FUNCTION_BLOCK FB_DiagnosisEtherCATSlaveWc2 IMPLEMENTS I_DiagnosisEtherCATSlave
VAR_INPUT
	sSlaveName					:STRING	:='NameNotSet';				//スレーブ名
END_VAR
VAR
	_bError						:BOOL;
	
	fbStateDiagnosis			:FB_StateDiagnosis;
	fbWcStateDiagnosis1			:FB_WcStateDiagnosis;
	fbWcStateDiagnosis2			:FB_WcStateDiagnosis;
END_VAR

(*エラー発生を出力*)
PROPERTY bError : BOOL
GET
bError:=_bError;
END_GET
END_PROPERTY

(*呼び出して診断実行*)
METHOD Execute
//診断用FBを呼び出し
fbStateDiagnosis(sSlaveName:=sSlaveName);
fbWcStateDiagnosis1(sSlaveName:=sSlaveName);
fbWcStateDiagnosis2(sSlaveName:=sSlaveName);

_bError:=fbStateDiagnosis.bError OR fbWcStateDiagnosis1.bError OR fbWcStateDiagnosis2.bError;
END_METHOD

END_FUNCTION_BLOCK

(* stored: Version 1.1.0.1
   POU FB_DiagnosisEtherCATSlaveWc2: Id {43d062e3-fee5-42c2-9ca9-d2a3a2982dac}, SpecialFunc None
   Property bError: Id {65139e7b-585f-4c34-9ae7-09df7cc57b61}
   Get Get: Id {3ec7d4f6-88ca-4377-9ea0-a8a8a53beebf}
   Method Execute: Id {0d918983-498a-4571-930d-74f126bea5ae} *)
